VAR_GLOBAL
	L_EinbruchBild : STRING;
	WetterBild : STRING := BildWolke;
END_VAR

(* stored: Version 1.1.0.1, ProductVersion 3.1.4018.5
   GVL Haus2: Id {864269e4-283e-4edd-b095-d41ed7564092} *)
